TYPE ST_DLK_Zustand :
STRUCT
	Betrieb				: BOOL;

	Leistung_elek			: REAL;	(* W *)
	Energie_elek			: REAL;
	Drehzahl				: REAL;	(* U/min *)
	Zeit_Betrieb			: INT;	(* h *)
	Druck_Auslass		: REAL;
	Temp_Umgebung		: REAL;
	Temp_Vorlauf		: REAL;
	Temp_Ruecklauf		: REAL;
	Modul_Meld_Code1	: WORD;
	Modul_Meld_Code2	: WORD;


	Betriebsstunden			: DWORD;
	Kompressorauslass_bar	: REAL;
	Druckluftmenge_erzeugt	: REAL;
	Drucktaupunkt			: REAL;
	Elementauslass			: REAL;
	Maschinenstatus			: BYTE;

	Stoerung				: BOOL;
	Stoerung_Code		: WORD;

	Warnung				: BOOL;
	Warnung_Code		: WORD;

	Status				: SINT;

	Quittierung			: BOOL;


END_STRUCT
END_TYPE

(* stored: Version 1.1.0.1, ProductVersion 3.1.4024.9
   DUT ST_DLK_Zustand: Id {29b8befe-5f20-419b-9ffc-eeb85a562c65} *)
